FUNCTION_BLOCK FBlock (* Basic function block *)
  (* Standard: 61499 *)
  (* Version 1.0, 11/20/2015 9:00 AM, Kawsihen, Kawsihen_s Macintosh *)
  (* Compiler header: package mypackage *)
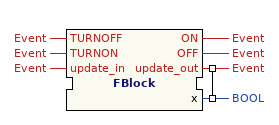
  EVENT_INPUT
    TURNOFF;
    TURNON;
    update_in;
  END_EVENT
  EVENT_OUTPUT
    ON;
    OFF;
    update_out WITH x;
  END_EVENT
  VAR_OUTPUT
    x : BOOL;
  END_VAR
  VAR
    k : REAL;
    d : REAL;
    signal_u : REAL;
    signal : REAL;
    y : REAL;
    C1y : REAL;
  END_VAR
  EC_STATES
    Start : init;
    b1 : b1Algo;
    b2 : b2Algo;
    b3 : b3Algo;
    b4 : b4Algo;
    t_state1 : t_state1Algo;
    t_state2 : t_state2Algo;
    t_state3 : t_state3Algo;
    t_state4 : t_state4Algo;
  END_STATES
  EC_TRANSITIONS
    Start TO b1 := True;
    b1 TO t_state1 := TURNON;
    t_state1 TO b2 := True;
    b2 TO t_state2 := true &&  (y >= 0.1);
    t_state2 TO b3 := True;
    b3 TO t_state3 := TURNOFF;
    t_state3 TO b4 := True;
    b4 TO t_state4 := true &&  (y >= 0.1);
    t_state4 TO b1 := True;
    b1 TO b1 := y >= 0 && y <= 0;
    b2 TO b2 := y < 0.1;
    b3 TO b3 := y >= 0 && y <= 0;
    b4 TO b4 := y < 0.1;
  END_TRANSITIONS
  ALGORITHM b1Algo IN C:
me->C1y = 0;
me->y = (float) me->C1y;
me->k++;
  END_ALGORITHM
  ALGORITHM b2Algo IN C:
me->C1y = 0;
me->y = (float) me->C1y + me->d*me->k;
me->k++;
  END_ALGORITHM
  ALGORITHM b3Algo IN C:
me->C1y = 0;
me->y = (float) me->C1y;
me->k++;
  END_ALGORITHM
  ALGORITHM b4Algo IN C:
me->C1y = 0;
me->y = (float) me->C1y + me->d*me->k;
me->k++;
  END_ALGORITHM
  ALGORITHM init IN C:
me->d = 0.01;
me->k = 0;
;
  END_ALGORITHM
  ALGORITHM t_state1Algo IN C:
me->y = me->y;
me->k = 0;
  END_ALGORITHM
  ALGORITHM t_state2Algo IN C:
me->y = 0;
me->signal = 1;
me->k = 0;
  END_ALGORITHM
  ALGORITHM t_state3Algo IN C:
me->y = me->y;
me->k = 0;
  END_ALGORITHM
  ALGORITHM t_state4Algo IN C:
me->y = 0;
me->signal = 0;
me->k = 0;
  END_ALGORITHM
END_FUNCTION_BLOCK
